(* Logix 5000 project; controller IF2_DEMO Emulate 5570 rev 20.12; software revision 20.04; part 8 of 8 *)
(* tags used below, declared in another part *)
   OrderQty : DINT[4];
   PartCountRollOver : DINT;
   RefillLine : LineData;
   Timer1000ms : TIMER;
   Timer250ms : TIMER;
   WallClock : DINT[7];
   WC : WC[10];

PROGRAM PackR   (* main routine MainRoutine *)
VAR
   ATest : BOOL;
   Block_Delay : TIMER := (PRE := 15000);
   Blocked_L : BOOL;
   BottleNum : STRING := '3';
   Ctrl_Bit : BOOL;
   DownStream_Run : BOOL := 1;
   DownStream_Running : BOOL := 1;   // Not used - no downstream wc
   Events : Events := (DownTime.Breakdown := 1, DownTime.BreakdownCode := 4, Control.StandbyCode := 1, Control.Auto := 1);
   Events_Control_Auto : ALIAS FOR WC_L.EventTrigger[0].5;
   Events_Control_OpStop : ALIAS FOR WC_L.EventTrigger[0].3;
   Events_Control_Run : ALIAS FOR WC_L.EventTrigger[0].1;
   Events_Control_Running : BOOL;
   Events_Control_Standby : ALIAS FOR WC_L.EventTrigger[0].0;
   Events_Control_StandbyCode : ALIAS FOR WC_L.EventValue_REAL[1];
   Events_DownTime_Breakdown : ALIAS FOR WC_L.EventTrigger[0].2;
   Events_DownTime_BreakdownCode : ALIAS FOR WC_L.EventValue_REAL[2];
   Events_DownTime_Testing : ALIAS FOR WC_L.EventTrigger[0].7;
   Events_DownTime_UnschedMaint : ALIAS FOR WC_L.EventTrigger[0].6;
   Events_Operate_Load : ALIAS FOR WC_L.EventTrigger[0].10;
   Events_Operate_OrderProc : ALIAS FOR WC_L.EventTrigger[0].11;
   Events_Operate_Setup : ALIAS FOR WC_L.EventTrigger[0].9;
   FillOunces : INT := 32;
   HMI : HMIVars := (ScrapRate := 5.0, SpeedControl := 90.0, PrevSpeed := 100.0, PartCountRollOver := 9999999, MfgTimeBase := 1, MaxEventDur := 21.0, MinEventDur := 9.0, EventsPerHr := 100, EventDur := 16.570301, RunDur := 18.429699, MinRunDur := 5.0);
   MfgOrders : MfgOrders := (CustomerName := 'Big-Mart', OrderName := 'A123', OrderQty := 30000, ProdRate := 60.0, PartName := 'STRAW-R40', WorkcellName := 'PackR', PartNameSav := 'STRAW-R40');
   MfgOrders_CustomerName : ALIAS FOR WC_L.FlexSTRING[4];
   MfgOrders_OrderName : ALIAS FOR WC_L.FlexSTRING[3];
   MfgOrders_PartName : ALIAS FOR WC_L.FlexSTRING[0];
   Motion : DINT := 53;
   Motion_Counter : DINT := 1;
   Motion_Speed : DINT := 12;
   MotionCount : TIMER := (PRE := 2400);
   OEE : OEE := (IdealCycleTime := 2.0, Parts.Total := 1051, Parts.Good := 998, Parts.Scrap := 53);
   OEE_IdealCycleTime : ALIAS FOR WC_L.IdealCT;
   OEE_Parts_Good : ALIAS FOR WC_L.GoodParts;
   OEE_Parts_Scrap : ALIAS FOR WC_L.ScrapParts;
   OEE_Parts_Total : ALIAS FOR WC_L.TotalParts;
   onsbits : DINT;
   OperatorID : ALIAS FOR WC_L.FlexREAL[1];
   Pressure1 : ALIAS FOR WC_L.PV[0];   // PSI
   ProductColorCode : INT;
   RecipeFlag : BOOL;
   RecipeName : STRING := 'Super';
   SIM : SimVars := (Run.PRE := 18430, Event.PRE := 9000, Setup.PRE := 9000, EventNumber := 11, UtilityBool[2] := 1);
        .UTILITYBOOL[0]   // Enter Auto Mode ONS
        .UTILITYBOOL[1]   // Work Order Complete ONS
        .UTILITYBOOL[2]   // First Scan Bit
   Starve_Delay : TIMER := (PRE := 15000);
   Starved_L : BOOL;
   Suppress : Events;
   Temperature1 : ALIAS FOR WC_L.PV[1];   // DEG
   UpStream_Run : ALIAS FOR WC[5].EventTrigger[0].1;
   UpStream_Running : ALIAS FOR WC[5].EventTrigger[0].8;
   WC_L : ALIAS FOR WC[9];
END_VAR

ROUTINE MainRoutine   (* ladder *)
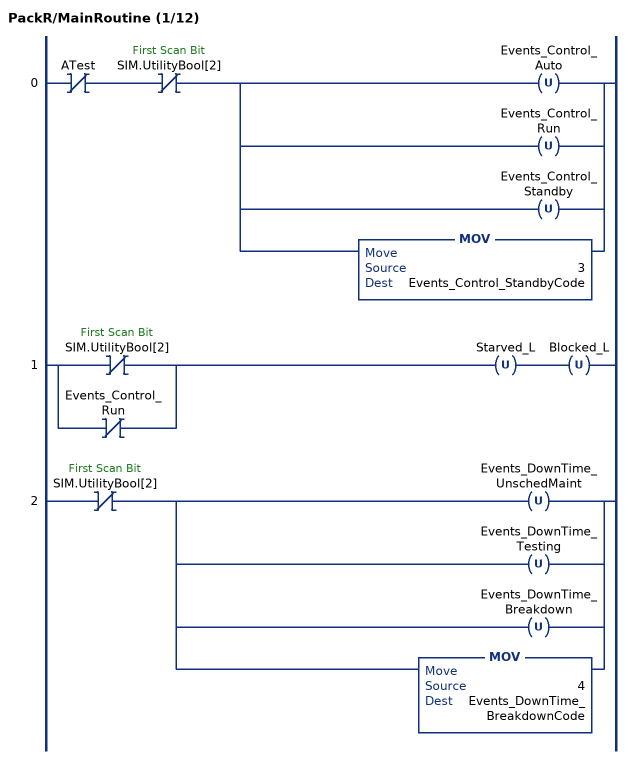
   0: XIO(ATest)XIO(SIM.UtilityBool[2])[OTU(Events_Control_Auto) ,OTU(Events_Control_Run) ,OTU(Events_Control_Standby) ,MOV(3,Events_Control_StandbyCode) ];
   1: [XIO(SIM.UtilityBool[2]) ,XIO(Events_Control_Run) ]OTU(Starved_L)OTU(Blocked_L);
   2: XIO(SIM.UtilityBool[2])[OTU(Events_DownTime_UnschedMaint) ,OTU(Events_DownTime_Testing) ,OTU(Events_DownTime_Breakdown) ,MOV(4,Events_DownTime_BreakdownCode) ];
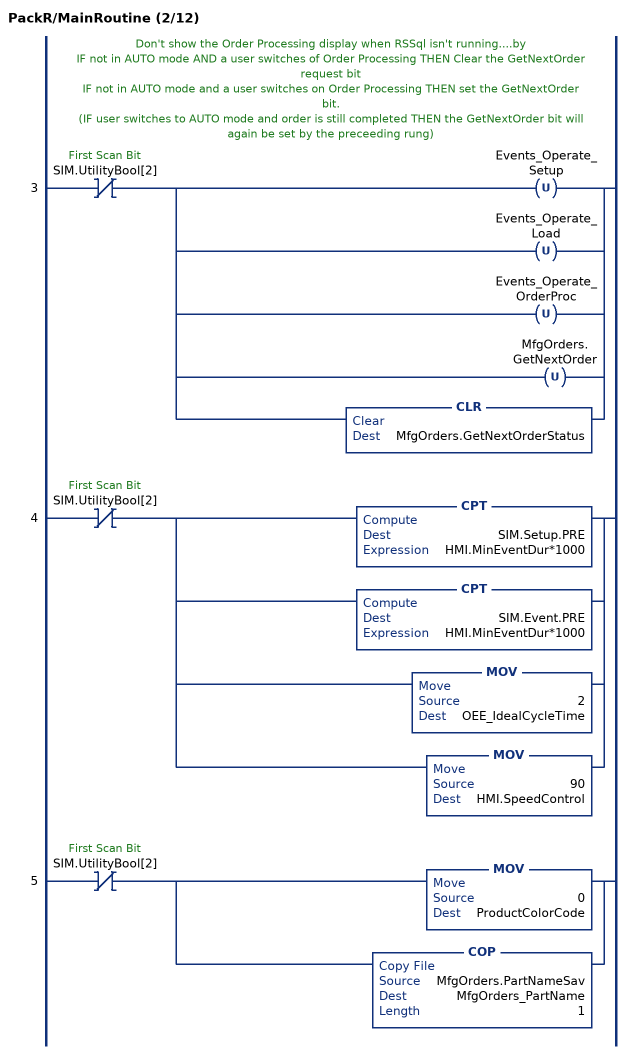
   // Don't show the Order Processing display when RSSql isn't running....by
   // IF not in AUTO mode AND a user switches of Order Processing THEN Clear the GetNextOrder request bit
   // IF not in AUTO mode and a user switches on Order Processing THEN set the GetNextOrder bit.
   // (IF user switches to AUTO mode and order is still completed THEN the GetNextOrder bit will again be set by the preceeding rung)
   3: XIO(SIM.UtilityBool[2])[OTU(Events_Operate_Setup) ,OTU(Events_Operate_Load) ,OTU(Events_Operate_OrderProc) ,OTU(MfgOrders.GetNextOrder) ,CLR(MfgOrders.GetNextOrderStatus) ];
   4: XIO(SIM.UtilityBool[2])[CPT(SIM.Setup.PRE,HMI.MinEventDur*1000) ,CPT(SIM.Event.PRE,HMI.MinEventDur*1000) ,MOV(2,OEE_IdealCycleTime) ,MOV(90,HMI.SpeedControl) ];
   5: XIO(SIM.UtilityBool[2])[MOV(0,ProductColorCode) ,COP(MfgOrders.PartNameSav,MfgOrders_PartName,1) ];
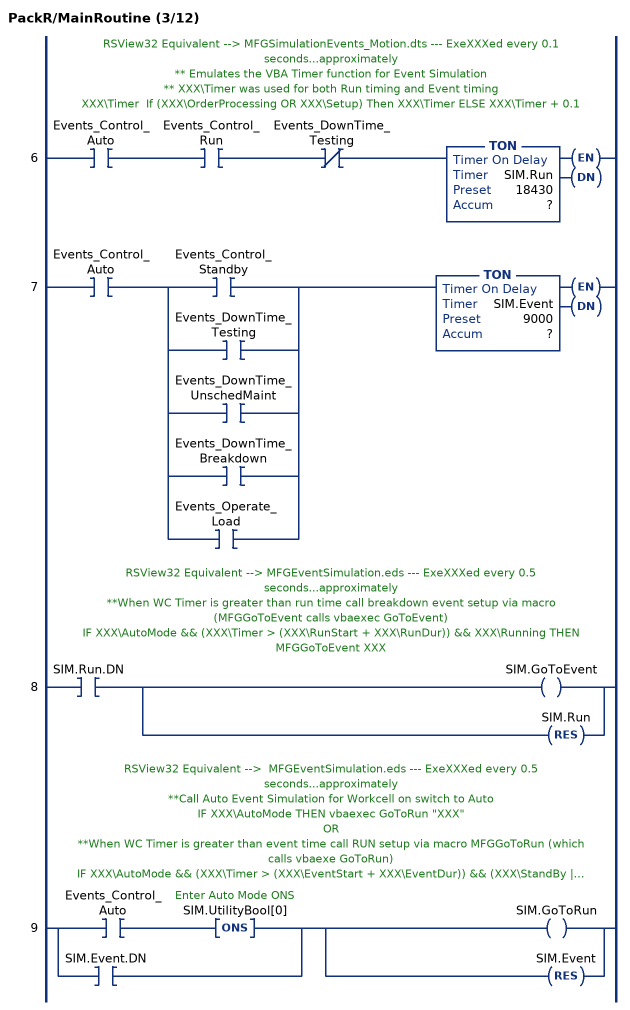
   // RSView32 Equivalent --> MFGSimulationEvents_Motion.dts --- ExeXXXed every 0.1 seconds...approximately
   // ** Emulates the VBA Timer function for Event Simulation
   // ** XXX\Timer was used for both Run timing and Event timing
   // XXX\Timer	If (XXX\OrderProcessing OR XXX\Setup) Then XXX\Timer ELSE XXX\Timer + 0.1
   6: XIC(Events_Control_Auto)XIC(Events_Control_Run)XIO(Events_DownTime_Testing)TON(SIM.Run,?,?);
   7: XIC(Events_Control_Auto)[XIC(Events_Control_Standby) ,XIC(Events_DownTime_Testing) ,XIC(Events_DownTime_UnschedMaint) ,XIC(Events_DownTime_Breakdown) ,XIC(Events_Operate_Load) ]TON(SIM.Event,?,?);
   // RSView32 Equivalent --> MFGEventSimulation.eds --- ExeXXXed every 0.5 seconds...approximately
   // **When WC Timer is greater than run time call breakdown event setup via macro (MFGGoToEvent calls vbaexec GoToEvent)
   // IF XXX\AutoMode && (XXX\Timer > (XXX\RunStart + XXX\RunDur)) && XXX\Running THEN MFGGoToEvent XXX
   8: XIC(SIM.Run.DN)[OTE(SIM.GoToEvent) ,RES(SIM.Run) ];
   // RSView32 Equivalent -->  MFGEventSimulation.eds --- ExeXXXed every 0.5 seconds...approximately
   // **Call Auto Event Simulation for Workcell on switch to Auto
   // IF XXX\AutoMode THEN vbaexec GoToRun "XXX"
   // OR
   // **When WC Timer is greater than event time call RUN setup via macro MFGGoToRun (which calls vbaexe GoToRun)
   // IF XXX\AutoMode && (XXX\Timer > (XXX\EventStart + XXX\EventDur)) && (XXX\StandBy || XXX\Test || XXX\UnSchedMaint || XXX\Breakdown ||XXX\Load) THEN MFGGoToRun XXX
   9: [XIC(Events_Control_Auto) ONS(SIM.UtilityBool[0]) ,XIC(SIM.Event.DN) ][OTE(SIM.GoToRun) ,RES(SIM.Event) ];
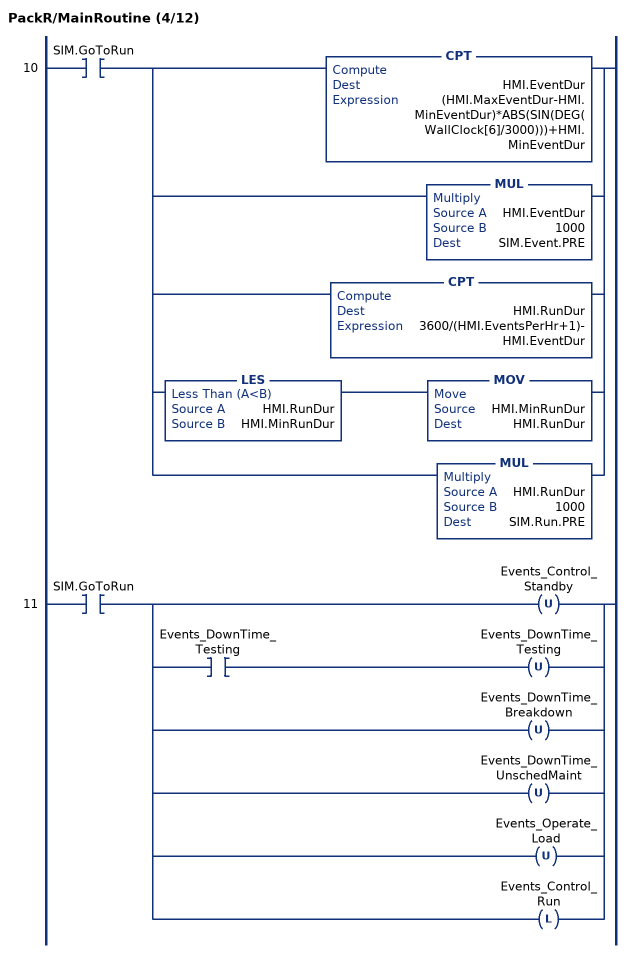
   10: XIC(SIM.GoToRun)[CPT(HMI.EventDur,(HMI.MaxEventDur-HMI.MinEventDur)*ABS(SIN(DEG(WallClock[6]/3000)))+HMI.MinEventDur) ,MUL(HMI.EventDur,1000,SIM.Event.PRE) ,CPT(HMI.RunDur,3600/(HMI.EventsPerHr+1)-HMI.EventDur) ,LES(HMI.RunDur,HMI.MinRunDur) MOV(HMI.MinRunDur,HMI.RunDur) ,MUL(HMI.RunDur,1000,SIM.Run.PRE) ];
   11: XIC(SIM.GoToRun)[OTU(Events_Control_Standby) ,XIC(Events_DownTime_Testing) OTU(Events_DownTime_Testing) ,OTU(Events_DownTime_Breakdown) ,OTU(Events_DownTime_UnschedMaint) ,OTU(Events_Operate_Load) ,OTL(Events_Control_Run) ];
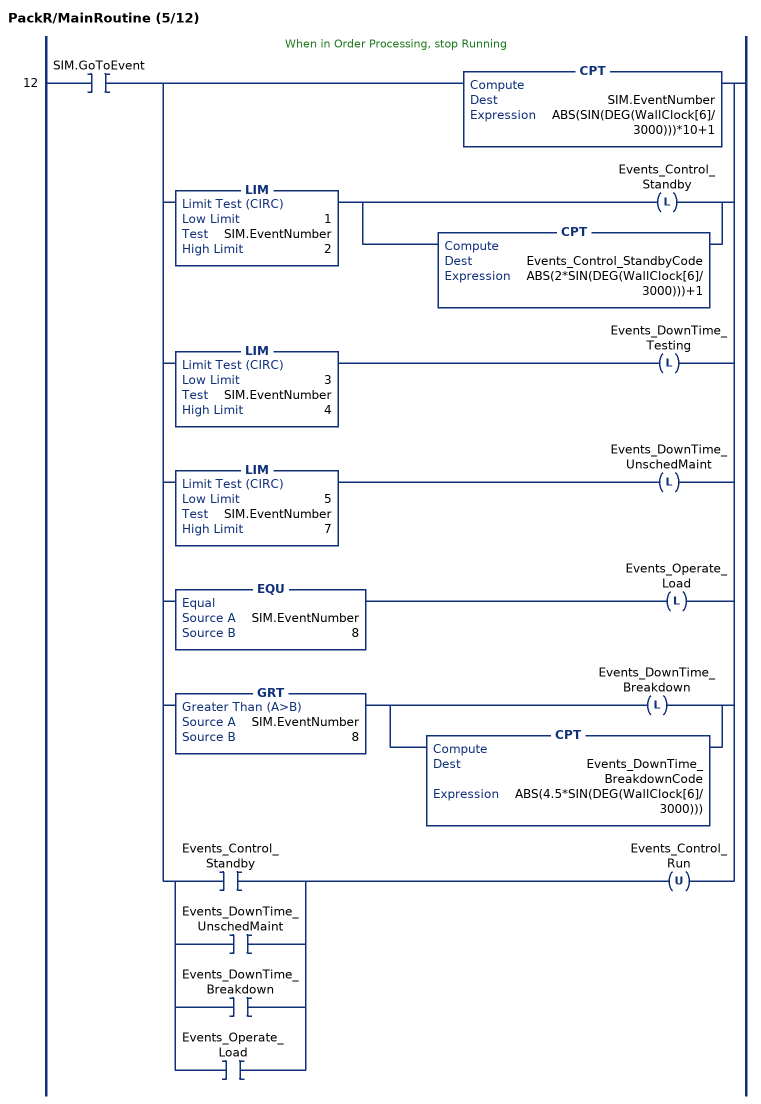
   // When in Order Processing, stop Running
   12: XIC(SIM.GoToEvent)[CPT(SIM.EventNumber,ABS(SIN(DEG(WallClock[6]/3000)))*10+1) ,LIM(1,SIM.EventNumber,2) [OTL(Events_Control_Standby) ,CPT(Events_Control_StandbyCode,ABS(2*SIN(DEG(WallClock[6]/3000)))+1) ] ,LIM(3,SIM.EventNumber,4) OTL(Events_DownTime_Testing) ,LIM(5,SIM.EventNumber,7) OTL(Events_DownTime_UnschedMaint) ,EQU(SIM.EventNumber,8) OTL(Events_Operate_Load) ,GRT(SIM.EventNumber,8) [OTL(Events_DownTime_Breakdown) ,CPT(Events_DownTime_BreakdownCode,ABS(4.5*SIN(DEG(WallClock[6]/3000)))) ] ,[XIC(Events_Control_Standby) ,XIC(Events_DownTime_UnschedMaint) ,XIC(Events_DownTime_Breakdown) ,XIC(Events_Operate_Load) ] OTU(Events_Control_Run) ];
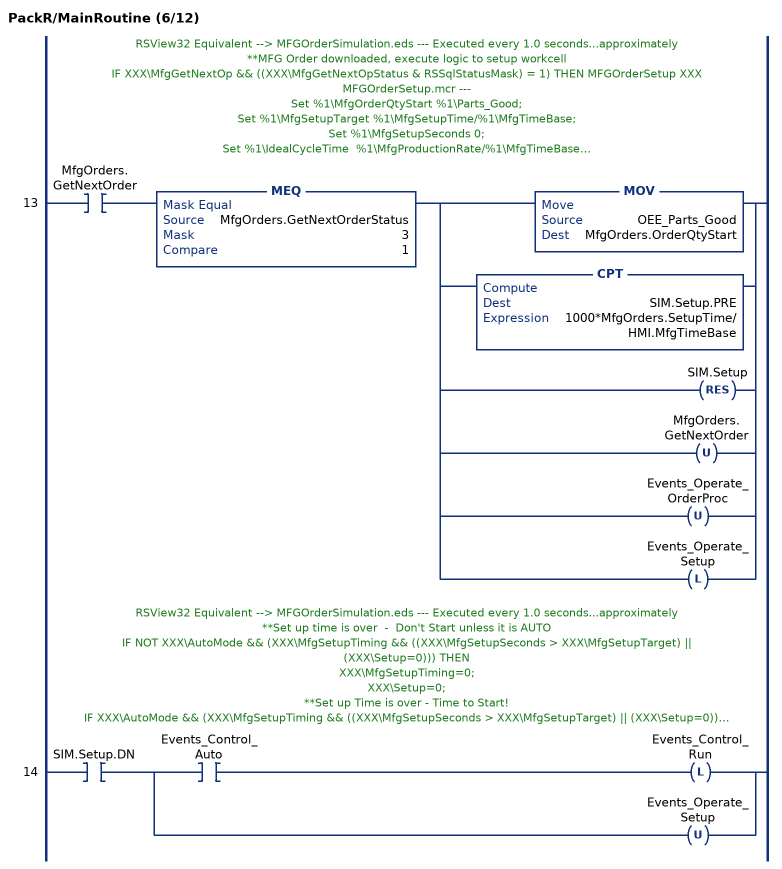
   // RSView32 Equivalent --> MFGOrderSimulation.eds --- Executed every 1.0 seconds...approximately
   // **MFG Order downloaded, execute logic to setup workcell
   // IF XXX\MfgGetNextOp && ((XXX\MfgGetNextOpStatus & RSSqlStatusMask) = 1) THEN MFGOrderSetup XXX
   // MFGOrderSetup.mcr ---
   // 	Set %1\MfgOrderQtyStart %1\Parts_Good;
   // 	Set %1\MfgSetupTarget %1\MfgSetupTime/%1\MfgTimeBase;
   // 	Set %1\MfgSetupSeconds 0;
   // 	Set %1\IdealCycleTime  %1\MfgProductionRate/%1\MfgTimeBase;
   // 	Set %1\MfgGetNextOp 0;
   // 	Set %1\Setup 1;
   // 	Set %1\OrderProcessing 0;
   // 	Set %1\MfgSetupTiming 1;
   13: XIC(MfgOrders.GetNextOrder)MEQ(MfgOrders.GetNextOrderStatus,3,1)[MOV(OEE_Parts_Good,MfgOrders.OrderQtyStart) ,CPT(SIM.Setup.PRE,1000*MfgOrders.SetupTime/HMI.MfgTimeBase) ,RES(SIM.Setup) ,OTU(MfgOrders.GetNextOrder) ,OTU(Events_Operate_OrderProc) ,OTL(Events_Operate_Setup) ];
   // RSView32 Equivalent --> MFGOrderSimulation.eds --- Executed every 1.0 seconds...approximately
   // **Set up time is over  -  Don't Start unless it is AUTO
   // IF NOT XXX\AutoMode && (XXX\MfgSetupTiming && ((XXX\MfgSetupSeconds > XXX\MfgSetupTarget) || (XXX\Setup=0))) THEN
   // 	XXX\MfgSetupTiming=0;
   // 	XXX\Setup=0;
   // **Set up Time is over - Time to Start!
   // IF XXX\AutoMode && (XXX\MfgSetupTiming && ((XXX\MfgSetupSeconds > XXX\MfgSetupTarget) || (XXX\Setup=0))) THEN
   // 	XXX\MfgSetupTiming=0;
   // 	XXX\Setup=0;
   // 	XXX\RUNNING=1
   14: XIC(SIM.Setup.DN)[XIC(Events_Control_Auto) OTL(Events_Control_Run) ,OTU(Events_Operate_Setup) ];
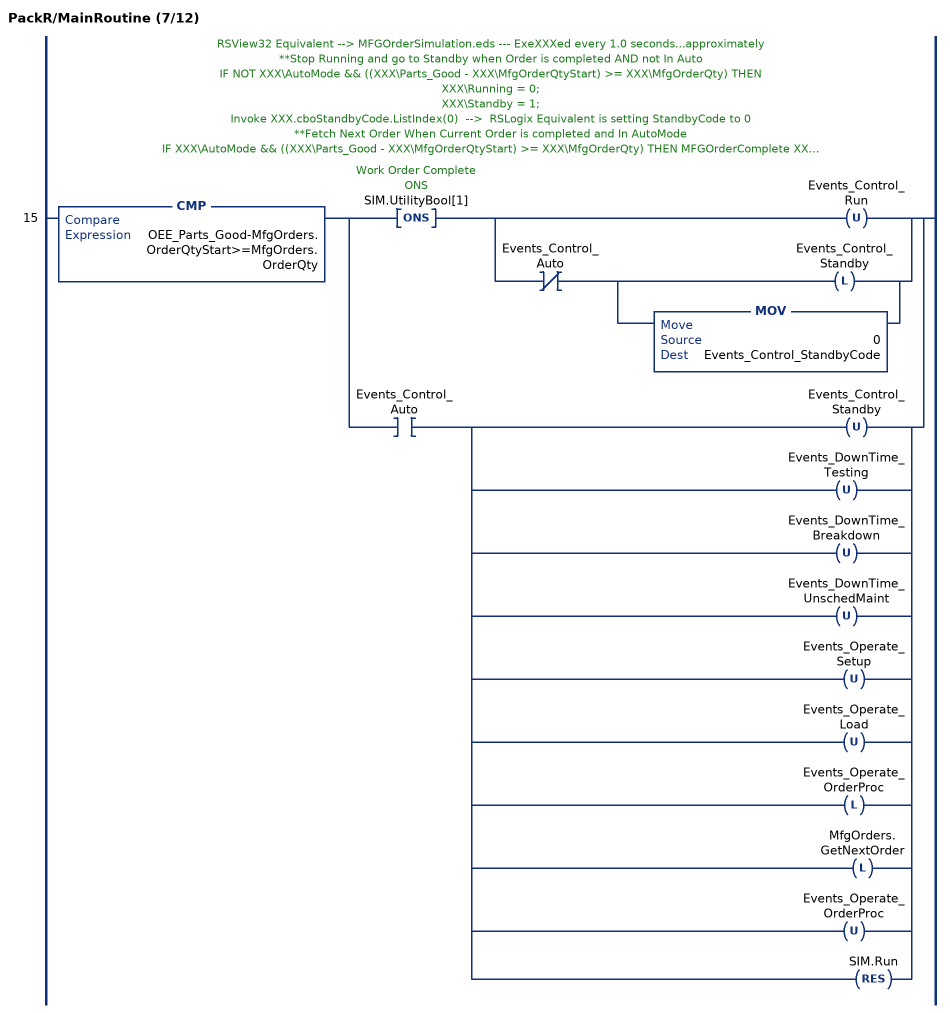
   // RSView32 Equivalent --> MFGOrderSimulation.eds --- ExeXXXed every 1.0 seconds...approximately
   // **Stop Running and go to Standby when Order is completed AND not In Auto
   // IF NOT XXX\AutoMode && ((XXX\Parts_Good - XXX\MfgOrderQtyStart) >= XXX\MfgOrderQty) THEN
   // 	XXX\Running = 0;
   // 	XXX\Standby = 1;
   // 	Invoke XXX.cboStandbyCode.ListIndex(0)  -->  RSLogix Equivalent is setting StandbyCode to 0
   // **Fetch Next Order When Current Order is completed and In AutoMode
   // IF XXX\AutoMode && ((XXX\Parts_Good - XXX\MfgOrderQtyStart) >= XXX\MfgOrderQty) THEN MFGOrderComplete XXX
   // MFGOrderComplete.mcr --- (Macros exeXXXed when called. %1 is the Workcell name -- typical all mcrs)
   // 	Set %1\RunStart %1\Timer;
   // 	Set %1\StandBy 0;
   // 	Set %1\Test 0;
   // 	Set %1\UnSchedMaint 0;
   // 	Set %1\Breakdown 0;
   // 	Set %1\Load 0;
   // 	Set %1\OrderProcessing 1;
   // 	Set %1\Running 0;
   // 	Set %1\MFGGetNextOpStatus 0;
   // 	Set %1\MFGGetNextOp 1
   15: CMP(OEE_Parts_Good-MfgOrders.OrderQtyStart>=MfgOrders.OrderQty)[ONS(SIM.UtilityBool[1]) [OTU(Events_Control_Run) ,XIO(Events_Control_Auto) [OTL(Events_Control_Standby) ,MOV(0,Events_Control_StandbyCode) ] ] ,XIC(Events_Control_Auto) [OTU(Events_Control_Standby) ,OTU(Events_DownTime_Testing) ,OTU(Events_DownTime_Breakdown) ,OTU(Events_DownTime_UnschedMaint) ,OTU(Events_Operate_Setup) ,OTU(Events_Operate_Load) ,OTL(Events_Operate_OrderProc) ,OTL(MfgOrders.GetNextOrder) ,OTU(Events_Operate_OrderProc) ,RES(SIM.Run) ] ];
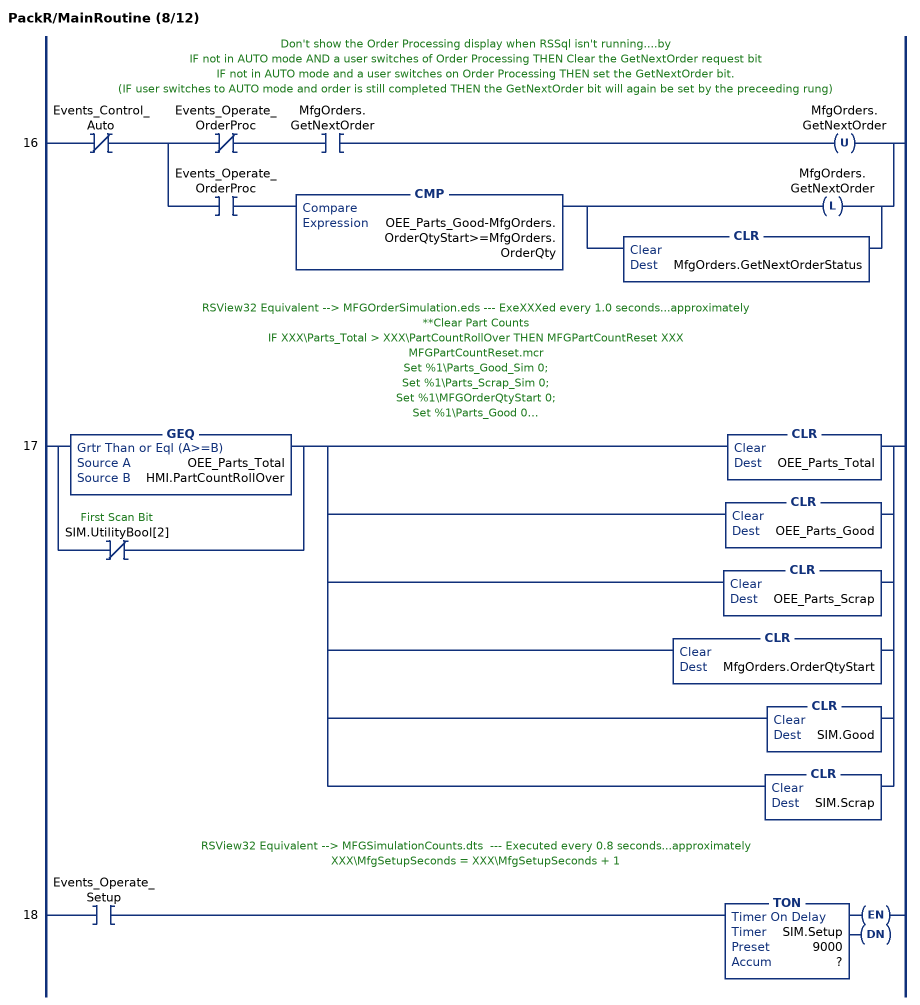
   // Don't show the Order Processing display when RSSql isn't running....by
   // IF not in AUTO mode AND a user switches of Order Processing THEN Clear the GetNextOrder request bit
   // IF not in AUTO mode and a user switches on Order Processing THEN set the GetNextOrder bit.
   // (IF user switches to AUTO mode and order is still completed THEN the GetNextOrder bit will again be set by the preceeding rung)
   16: XIO(Events_Control_Auto)[XIO(Events_Operate_OrderProc) XIC(MfgOrders.GetNextOrder) OTU(MfgOrders.GetNextOrder) ,XIC(Events_Operate_OrderProc) CMP(OEE_Parts_Good-MfgOrders.OrderQtyStart>=MfgOrders.OrderQty) [OTL(MfgOrders.GetNextOrder) ,CLR(MfgOrders.GetNextOrderStatus) ] ];
   // RSView32 Equivalent --> MFGOrderSimulation.eds --- ExeXXXed every 1.0 seconds...approximately
   // **Clear Part Counts
   // IF XXX\Parts_Total > XXX\PartCountRollOver THEN MFGPartCountReset XXX
   // MFGPartCountReset.mcr
   // 	Set %1\Parts_Good_Sim 0;
   // 	Set %1\Parts_Scrap_Sim 0;
   // 	Set %1\MFGOrderQtyStart 0;
   // 	Set %1\Parts_Good 0;
   // 	Set %1\Parts_Scrap 0;
   // 	Set %1\Parts_Total 0
   17: [GEQ(OEE_Parts_Total,HMI.PartCountRollOver) ,XIO(SIM.UtilityBool[2]) ][CLR(OEE_Parts_Total) ,CLR(OEE_Parts_Good) ,CLR(OEE_Parts_Scrap) ,CLR(MfgOrders.OrderQtyStart) ,CLR(SIM.Good) ,CLR(SIM.Scrap) ];
   // RSView32 Equivalent --> MFGSimulationCounts.dts	--- Executed every 0.8 seconds...approximately
   // XXX\MfgSetupSeconds = XXX\MfgSetupSeconds + 1
   18: XIC(Events_Operate_Setup)TON(SIM.Setup,?,?);
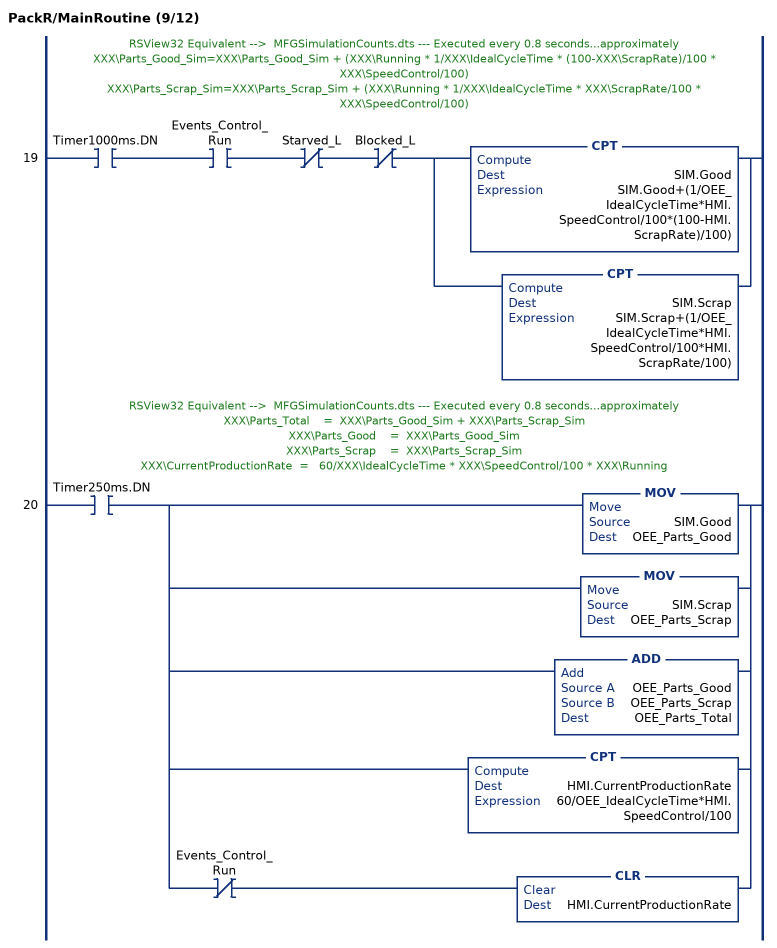
   // RSView32 Equivalent -->  MFGSimulationCounts.dts --- Executed every 0.8 seconds...approximately
   // XXX\Parts_Good_Sim=XXX\Parts_Good_Sim + (XXX\Running * 1/XXX\IdealCycleTime * (100-XXX\ScrapRate)/100 * XXX\SpeedControl/100)
   // XXX\Parts_Scrap_Sim=XXX\Parts_Scrap_Sim + (XXX\Running * 1/XXX\IdealCycleTime * XXX\ScrapRate/100 * XXX\SpeedControl/100)
   19: XIC(Timer1000ms.DN)XIC(Events_Control_Run)XIO(Starved_L)XIO(Blocked_L)[CPT(SIM.Good,SIM.Good+(1/OEE_IdealCycleTime*HMI.SpeedControl/100*(100-HMI.ScrapRate)/100)) ,CPT(SIM.Scrap,SIM.Scrap+(1/OEE_IdealCycleTime*HMI.SpeedControl/100*HMI.ScrapRate/100)) ];
   // RSView32 Equivalent -->  MFGSimulationCounts.dts --- Executed every 0.8 seconds...approximately
   // XXX\Parts_Total		=	XXX\Parts_Good_Sim + XXX\Parts_Scrap_Sim
   // XXX\Parts_Good		=	XXX\Parts_Good_Sim
   // XXX\Parts_Scrap		=	XXX\Parts_Scrap_Sim
   // XXX\CurrentProductionRate  = 	60/XXX\IdealCycleTime * XXX\SpeedControl/100 * XXX\Running
   20: XIC(Timer250ms.DN)[[MOV(SIM.Good,OEE_Parts_Good) ,MOV(SIM.Scrap,OEE_Parts_Scrap) ,ADD(OEE_Parts_Good,OEE_Parts_Scrap,OEE_Parts_Total) ] ,CPT(HMI.CurrentProductionRate,60/OEE_IdealCycleTime*HMI.SpeedControl/100) ,XIO(Events_Control_Run) CLR(HMI.CurrentProductionRate) ];
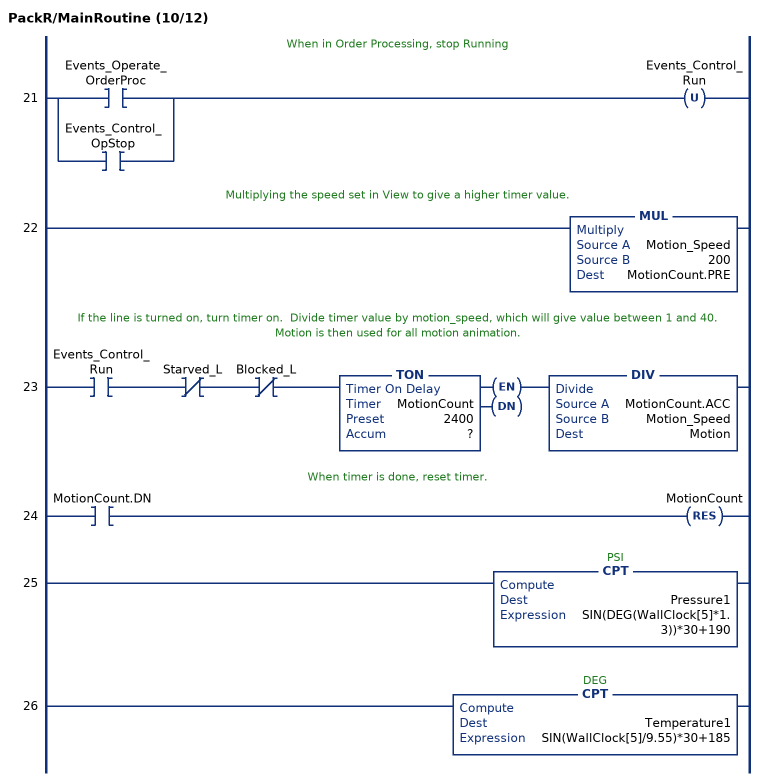
   // When in Order Processing, stop Running
   21: [XIC(Events_Operate_OrderProc) ,XIC(Events_Control_OpStop) ]OTU(Events_Control_Run);
   // Multiplying the speed set in View to give a higher timer value.
   22: MUL(Motion_Speed,200,MotionCount.PRE);
   // If the line is turned on, turn timer on.  Divide timer value by motion_speed, which will give value between 1 and 40.  Motion is then used for all motion animation.
   23: XIC(Events_Control_Run)XIO(Starved_L)XIO(Blocked_L)TON(MotionCount,?,?)DIV(MotionCount.ACC,Motion_Speed,Motion);
   // When timer is done, reset timer.
   24: XIC(MotionCount.DN)RES(MotionCount);
   25: CPT(Pressure1,SIN(DEG(WallClock[5]*1.3))*30+190);
   26: CPT(Temperature1,SIN(WallClock[5]/9.55)*30+185);
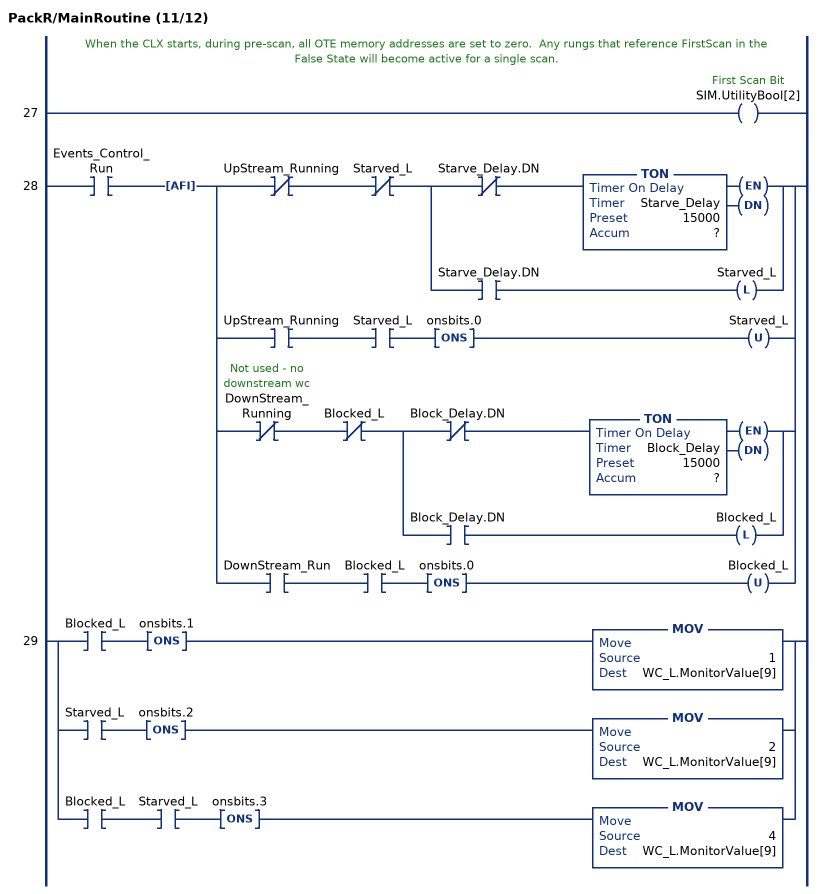
   // When the CLX starts, during pre-scan, all OTE memory addresses are set to zero.  Any rungs that reference FirstScan in the False State will become active for a single scan.
   27: OTE(SIM.UtilityBool[2]);
   28: XIC(Events_Control_Run)AFI()[[XIO(UpStream_Running) XIO(Starved_L) [XIO(Starve_Delay.DN) TON(Starve_Delay,?,?) ,XIC(Starve_Delay.DN) OTL(Starved_L) ] ,XIC(UpStream_Running) XIC(Starved_L) ONS(onsbits.0) OTU(Starved_L) ] ,[XIO(DownStream_Running) XIO(Blocked_L) [XIO(Block_Delay.DN) TON(Block_Delay,?,?) ,XIC(Block_Delay.DN) OTL(Blocked_L) ] ,XIC(DownStream_Run) XIC(Blocked_L) ONS(onsbits.0) OTU(Blocked_L) ] ];
   29: [XIC(Blocked_L) ONS(onsbits.1) MOV(1,WC_L.MonitorValue[9]) ,XIC(Starved_L) ONS(onsbits.2) MOV(2,WC_L.MonitorValue[9]) ,XIC(Blocked_L) XIC(Starved_L) ONS(onsbits.3) MOV(4,WC_L.MonitorValue[9]) ];
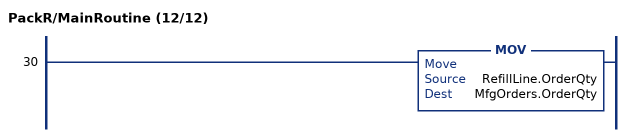
   30: MOV(RefillLine.OrderQty,MfgOrders.OrderQty);
END_ROUTINE
END_PROGRAM
